(* PLC project CoDeSys External Library Template, WAGO e!COCKPIT e!COCKPIT, author 3S - Smart Software Solutions GmbH *)
(* stored: creationDateTime 2019-10-29T12:37:19.5873699, version 3.5.5.30, modificationDateTime 2019-10-29T12:36:39.3744516, organization 3S - Smart Software Solutions GmbH *)
(* Library project template with all possible element types, docu and a sample project structure *)

TYPE ZADAJNIK_FCP : STRUCT
  sIdInstancji : STRING;
  rTemperaturaNastawiona : REAL;
  rTemperaturaPomieszczenia : REAL;
  rTemperaturaBazowaHMI : REAL := 293.15;
  rSkalaPotencjometruAutonomizacja : REAL := 1;
  rTemperaturaBazowaAutoAutonomizacja : REAL := 293.15;
  intTrybPracy : INT;
  xBrakKomunikacjiIZE : BOOL;
  xBrakKomunikacjiPLC : BOOL;
  xPokazPanelHMI : BOOL := TRUE;
  intTrybPracyHMI : INT := 1;
  xAutonomizacja : BOOL;
  sEnOceanIDodczytany : STRING;
  wCzasOdOstatniegoKomunikatu : WORD;
  xZwiekszTemperature : BOOL;
  xZmniejszTemperature : BOOL;
END_STRUCT;
END_TYPE
